EC00811=-138.9583,0.0000
EC00812=-136.5366,0.0000
EC00813=-135.0000,0.0000
EC00814=-133.4634,0.0000
EC00815=-131.0417,0.0000
EC00816=-127.9674,0.0000
EC00817=-127.2322,0.0000
EC00818=-127.3085,0.0000
EC00819=-127.4027,0.0000
EC00820=-127.4553,0.0000
EC00821=-127.3659,0.0000
EC00822=-125.6434,0.0000
EC00823=-122.6119,0.0000
EC00824=-118.7938,0.0000
EC00825=-114.6278,0.0000
EC00826=-110.3718,0.0000
EC00827=-106.2065,0.0000
EC00828=-102.3884,0.0000
EC00829=-99.3569,0.0000
EC00830=-97.6343,0.0000
EC00831=-97.5446,0.0000
EC00832=-97.5966,0.0000
EC00833=-97.6919,0.0000
EC00834=-97.7683,0.0000
EC00835=-97.0327,0.0000
EC00836=-93.9586,0.0000
EC00837=-91.5376,0.0000
EC00838=-90.0000,0.0000
EC00839=-88.4635,0.0000
EC00840=-86.0414,0.0000
EC00841=-82.9673,0.0000
EC00842=-82.2317,0.0000
EC00843=-82.3081,0.0000
EC00844=-82.4034,0.0000
EC00845=-82.4554,0.0000
EC00846=-82.3657,0.0000
EC00847=-80.6431,0.0000
EC00848=-77.6116,0.0000
EC00849=-73.7935,0.0000
EC00850=-69.6282,0.0000
EC00851=-65.3722,0.0000
EC00852=-61.2062,0.0000
EC00853=-57.3881,0.0000
EC00854=-54.3566,0.0000
EC00855=-52.6341,0.0000
EC00856=-52.5447,0.0000
EC00857=-52.5973,0.0000
EC00858=-52.6915,0.0000
EC00859=-52.7678,0.0000
EC00860=-52.0326,0.0000
EC00861=-48.9583,0.0000
EC00862=-46.5366,0.0000
EC00863=-45.0000,0.0000
EC00864=-43.4634,0.0000
EC00865=-41.0417,0.0000
EC00866=-37.9674,0.0000
EC00867=-37.2322,0.0000
EC00868=-37.3085,0.0000
EC00869=-37.4027,0.0000
EC00870=-37.4553,0.0000
EC00871=-37.3659,0.0000
EC00872=-35.6434,0.0000
EC00873=-32.6119,0.0000
EC00874=-28.7938,0.0000
EC00875=-24.6278,0.0000
EC00876=-20.3718,0.0000
EC00877=-16.2065,0.0000
EC00878=-12.3884,0.0000
EC00879=-9.3569,0.0000
EC00880=-7.6343,0.0000
EC00881=-7.5446,0.0000
EC00882=-7.5966,0.0000
EC00883=-7.6919,0.0000
EC00884=-7.7683,0.0000
EC00885=-7.0327,0.0000
EC00886=-3.9586,0.0000
EC00887=-1.5365,0.0000
EC00888=0.0000,0.0000
EC00889=0.0000,0.0000
EC00890=1.4747,0.0000
EC00891=3.8756,0.0000
EC00892=6.9699,0.0000
EC00893=7.6906,0.0000
EC00894=7.6170,0.0000
EC00895=7.5429,0.0000
EC00896=7.5106,0.0000
EC00897=7.6094,0.0000
EC00898=9.3401,0.0000
EC00899=35.6602,0.0000
EC00900=37.3910,0.0000
EC00901=37.4898,0.0000
EC00902=37.4572,0.0000
EC00903=37.3834,0.0000
EC00904=37.3085,0.0000
EC00905=38.0296,0.0000
EC00906=41.1238,0.0000
EC00907=43.5256,0.0000
EC00908=45.0000,0.0000
EC00909=46.4744,0.0000
EC00910=48.8762,0.0000
EC00911=51.9704,0.0000
EC00912=52.6915,0.0000
EC00913=52.6166,0.0000
EC00914=52.5428,0.0000
EC00915=52.5102,0.0000
EC00916=52.6090,0.0000
EC00917=54.3398,0.0000
EC00918=80.6599,0.0000
EC00919=82.3906,0.0000
EC00920=82.4894,0.0000
EC00921=82.4571,0.0000
EC00922=82.3830,0.0000
EC00923=82.3094,0.0000
EC00924=83.0301,0.0000
EC00925=86.1244,0.0000
EC00926=88.5253,0.0000
EC00927=90.0000,0.0000
EC00928=91.4736,0.0000
EC00929=93.8767,0.0000
EC00930=96.9699,0.0000
EC00931=97.6906,0.0000
EC00932=97.6170,0.0000
EC00933=97.5429,0.0000
EC00934=97.5106,0.0000
EC00935=97.6094,0.0000
EC00936=99.3401,0.0000
EC00937=125.6602,0.0000
EC00938=127.3910,0.0000
EC00939=127.4898,0.0000
EC00940=127.4572,0.0000
EC00941=127.3834,0.0000
EC00942=127.3085,0.0000
EC00943=128.0296,0.0000
EC00944=131.1238,0.0000
EC00945=133.5256,0.0000
EC00946=135.0000,0.0000
EC00947=136.4744,0.0000
EC00948=138.8762,0.0000
EC00949=141.9704,0.0000
EC00950=142.6915,0.0000
EC00951=142.6166,0.0000
EC00952=142.5428,0.0000
EC00953=142.5102,0.0000
EC00954=142.6090,0.0000
EC00955=144.3398,0.0000
EC00956=170.6599,0.0000
EC00957=172.3906,0.0000
EC00958=172.4894,0.0000
EC00959=172.4571,0.0000
EC00960=172.3830,0.0000
EC00961=172.3094,0.0000
EC00962=173.0301,0.0000
EC00963=176.1244,0.0000
EC00964=178.5253,0.0000
EC00965=180.0000,0.0000
EC00966=180.0000,0.0000
EC00967=-178.5264,0.0000
EC00968=-176.1233,0.0000
EC00969=-173.0301,0.0000
EC00970=-172.3094,0.0000
EC00971=-172.3830,0.0000
EC00972=-172.4571,0.0000
EC00973=-172.4894,0.0000
EC00974=-172.3906,0.0000
EC00975=-170.6599,0.0000
EC00976=-144.3398,0.0000
EC00977=-142.6090,0.0000
EC00978=-142.5102,0.0000
EC00979=-142.5428,0.0000
EC00980=-142.6166,0.0000
EC00981=-142.6915,0.0000
EC00982=-141.9704,0.0000
EC00983=-138.8762,0.0000
EC00984=-136.4744,0.0000
EC00985=-135.0000,0.0000
EC00986=-133.5256,0.0000
EC00987=-131.1238,0.0000
EC00988=-128.0296,0.0000
EC00989=-127.3085,0.0000
EC00990=-127.3834,0.0000
EC00991=-127.4572,0.0000
EC00992=-127.4898,0.0000
EC00993=-127.3910,0.0000
EC00994=-125.6602,0.0000
EC00995=-99.3401,0.0000
EC00996=-97.6094,0.0000
EC00997=-97.5106,0.0000
EC00998=-97.5429,0.0000
EC00999=-97.6170,0.0000
EC01000=-97.6906,0.0000
EC01001=-96.9699,0.0000
EC01002=-93.8756,0.0000
EC01003=-91.4747,0.0000
EC01004=-90.0000,0.0000
EC01005=-88.5264,0.0000
EC01006=-86.1233,0.0000
EC01007=-83.0301,0.0000
EC01008=-82.3094,0.0000
EC01009=-82.3830,0.0000
EC01010=-82.4571,0.0000
EC01011=-82.4894,0.0000
EC01012=-82.3906,0.0000
EC01013=-80.6599,0.0000
EC01014=-54.3398,0.0000
EC01015=-52.6090,0.0000
EC01016=-52.5102,0.0000
EC01017=-52.5428,0.0000
EC01018=-52.6166,0.0000
EC01019=-52.6915,0.0000
EC01020=-51.9704,0.0000
EC01021=-48.8762,0.0000
EC01022=-46.4744,0.0000
EC01023=-45.0000,0.0000
EC01024=-43.5256,0.0000
EC01025=-41.1238,0.0000
EC01026=-38.0296,0.0000
EC01027=-37.3085,0.0000
EC01028=-37.3834,0.0000
EC01029=-37.4572,0.0000
EC01030=-37.4898,0.0000
EC01031=-37.3910,0.0000
EC01032=-35.6602,0.0000
EC01033=-9.3401,0.0000
EC01034=-7.6094,0.0000
EC01035=-7.5106,0.0000
EC01036=-7.5429,0.0000
EC01037=-7.6170,0.0000
EC01038=-7.6906,0.0000
EC01039=-6.9699,0.0000
EC01040=-3.8767,0.0000
EC01041=-1.4736,0.0000
EC01042=0.0000,0.0000
EC01043=0.0000,0.0000
EC01044=1.4165,0.0000
EC01045=3.7994,0.0000
EC01046=6.9134,0.0000
EC01047=7.6249,0.0000
EC01048=7.5584,0.0000
EC01049=7.5104,0.0000
EC01050=37.4901,0.0000
EC01051=37.4412,0.0000
EC01052=37.3752,0.0000
EC01053=38.0867,0.0000
EC01054=41.2006,0.0000
EC01055=43.5844,0.0000
EC01056=45.0000,0.0000
EC01057=46.4156,0.0000
EC01058=48.8001,0.0000
EC01059=51.9133,0.0000
EC01060=52.6248,0.0000
EC01061=52.5588,0.0000
EC01062=52.5099,0.0000
EC01063=82.4896,0.0000
EC01064=82.4416,0.0000
EC01065=82.3751,0.0000
EC01066=83.0866,0.0000
EC01067=86.2006,0.0000
EC01068=88.5835,0.0000
EC01069=90.0000,0.0000
EC01070=91.4153,0.0000
EC01071=93.8005,0.0000
EC01072=96.9134,0.0000
EC01073=97.6249,0.0000
EC01074=97.5584,0.0000
EC01075=97.5104,0.0000
EC01076=127.4901,0.0000
EC01077=127.4412,0.0000
EC01078=127.3752,0.0000
EC01079=128.0867,0.0000
EC01080=131.2006,0.0000
EC01081=133.5844,0.0000
EC01082=135.0000,0.0000
EC01083=136.4156,0.0000
EC01084=138.8001,0.0000
EC01085=141.9133,0.0000
EC01086=142.6248,0.0000
EC01087=142.5588,0.0000
EC01088=142.5099,0.0000
EC01089=172.4896,0.0000
EC01090=172.4416,0.0000
EC01091=172.3751,0.0000
EC01092=173.0866,0.0000
EC01093=176.2006,0.0000
EC01094=178.5835,0.0000
EC01095=180.0000,0.0000
EC01096=180.0000,0.0000
EC01097=-178.5847,0.0000
EC01098=-176.1995,0.0000
EC01099=-173.0866,0.0000
EC01100=-172.3751,0.0000
EC01101=-172.4416,0.0000
EC01102=-172.4896,0.0000
EC01103=-142.5099,0.0000
EC01104=-142.5588,0.0000
EC01105=-142.6248,0.0000
EC01106=-141.9133,0.0000
EC01107=-138.7994,0.0000
EC01108=-136.4156,0.0000
EC01109=-135.0000,0.0000
EC01110=-133.5844,0.0000
EC01111=-131.1999,0.0000
EC01112=-128.0867,0.0000
EC01113=-127.3752,0.0000
EC01114=-127.4412,0.0000
EC01115=-127.4901,0.0000
EC01116=-97.5104,0.0000
EC01117=-97.5584,0.0000
EC01118=-97.6249,0.0000
EC01119=-96.9134,0.0000
EC01120=-93.7994,0.0000
EC01121=-91.4165,0.0000
EC01122=-90.0000,0.0000
EC01123=-88.5847,0.0000
EC01124=-86.1995,0.0000
EC01125=-83.0866,0.0000
EC01126=-82.3751,0.0000
EC01127=-82.4416,0.0000
EC01128=-82.4896,0.0000
EC01129=-52.5099,0.0000
EC01130=-52.5588,0.0000
EC01131=-52.6248,0.0000
EC01132=-51.9133,0.0000
EC01133=-48.7994,0.0000
EC01134=-46.4156,0.0000
EC01135=-45.0000,0.0000
EC01136=-43.5844,0.0000
EC01137=-41.1999,0.0000
EC01138=-38.0867,0.0000
EC01139=-37.3752,0.0000
EC01140=-37.4412,0.0000
EC01141=-37.4901,0.0000
EC01142=-7.5104,0.0000
EC01143=-7.5584,0.0000
EC01144=-7.6249,0.0000
EC01145=-6.9134,0.0000
EC01146=-3.8005,0.0000
EC01147=-1.4153,0.0000
EC01148=0.0000,0.0000
EC01149=0.0000,0.0000
EC01150=1.3641,0.0000
EC01151=3.7307,0.0000
EC01152=6.8641,0.0000
EC01153=7.5707,0.0000
EC01154=7.5193,0.0000
EC01155=37.4799,0.0000
EC01156=37.4296,0.0000
EC01157=38.1360,0.0000
EC01158=41.2692,0.0000
EC01159=43.6362,0.0000
EC01160=45.0000,0.0000
EC01161=46.3630,0.0000
EC01162=48.7308,0.0000
EC01163=51.8640,0.0000
EC01164=52.5704,0.0000
EC01165=52.5201,0.0000
EC01166=82.4807,0.0000
EC01167=82.4293,0.0000
EC01168=83.1359,0.0000
EC01169=86.2693,0.0000
EC01170=88.6359,0.0000
EC01171=90.0000,0.0000
EC01172=91.3630,0.0000
EC01173=93.7318,0.0000
EC01174=96.8641,0.0000
EC01175=97.5707,0.0000
EC01176=97.5193,0.0000
EC01177=127.4799,0.0000
EC01178=127.4296,0.0000
EC01179=128.1360,0.0000
EC01180=131.2692,0.0000
EC01181=133.6362,0.0000
EC01182=135.0000,0.0000
EC01183=136.3630,0.0000
EC01184=138.7308,0.0000
EC01185=141.8640,0.0000
EC01186=142.5704,0.0000
EC01187=142.5201,0.0000
EC01188=172.4807,0.0000
EC01189=172.4293,0.0000
EC01190=173.1359,0.0000
EC01191=176.2693,0.0000
EC01192=178.6359,0.0000
EC01193=180.0000,0.0000
EC01194=180.0000,0.0000
EC01195=-178.6370,0.0000
EC01196=-176.2682,0.0000
EC01197=-173.1359,0.0000
EC01198=-172.4293,0.0000
EC01199=-172.4807,0.0000
EC01200=-142.5201,0.0000
EC01201=-142.5704,0.0000
EC01202=-141.8640,0.0000
EC01203=-138.7308,0.0000
EC01204=-136.3638,0.0000
EC01205=-135.0000,0.0000
EC01206=-133.6370,0.0000
EC01207=-131.2692,0.0000
EC01208=-128.1360,0.0000
EC01209=-127.4296,0.0000
EC01210=-127.4799,0.0000
EC01211=-97.5193,0.0000
EC01212=-97.5707,0.0000
EC01213=-96.8641,0.0000
EC01214=-93.7307,0.0000
EC01215=-91.3641,0.0000
EC01216=-90.0000,0.0000
EC01217=-88.6370,0.0000
EC01218=-86.2682,0.0000
EC01219=-83.1359,0.0000
EC01220=-82.4293,0.0000
EC01221=-82.4807,0.0000
EC01222=-52.5201,0.0000
EC01223=-52.5704,0.0000
EC01224=-51.8640,0.0000
EC01225=-48.7308,0.0000
EC01226=-46.3638,0.0000
EC01227=-45.0000,0.0000
EC01228=-43.6370,0.0000
EC01229=-41.2692,0.0000
EC01230=-38.1360,0.0000
EC01231=-37.4296,0.0000
EC01232=-37.4799,0.0000
EC01233=-7.5193,0.0000
EC01234=-7.5707,0.0000
EC01235=-6.8641,0.0000
EC01236=-3.7318,0.0000
EC01237=-1.3630,0.0000
EC01238=0.0000,0.0000
EC01239=0.0000,0.0000
EC01240=1.3191,0.0000
EC01241=3.6720,0.0000
EC01242=6.8225,0.0000
EC01243=7.5303,0.0000
EC01244=7.5014,0.0000
EC01245=37.4983,0.0000
EC01246=37.4688,0.0000
EC01247=38.1772,0.0000
EC01248=41.3279,0.0000
EC01249=43.6816,0.0000
EC01250=45.0000,0.0000
EC01251=46.3184,0.0000
EC01252=48.6728,0.0000
EC01253=51.8228,0.0000
EC01254=52.5312,0.0000
EC01255=52.5017,0.0000
EC01256=82.4986,0.0000
EC01257=82.4697,0.0000
EC01258=83.1775,0.0000
EC01259=86.3280,0.0000
EC01260=88.6809,0.0000
EC01261=90.0000,0.0000
EC01262=91.3180,0.0000
EC01263=93.6719,0.0000
EC01264=96.8225,0.0000
EC01265=97.5303,0.0000
EC01266=97.5014,0.0000
EC01267=127.4983,0.0000
EC01268=127.4688,0.0000
EC01269=128.1772,0.0000
EC01270=131.3279,0.0000
EC01271=133.6816,0.0000
EC01272=135.0000,0.0000
EC01273=136.3184,0.0000
EC01274=138.6728,0.0000
EC01275=141.8228,0.0000
EC01276=142.5312,0.0000
EC01277=142.5017,0.0000
EC01278=172.4986,0.0000
EC01279=172.4697,0.0000
EC01280=173.1775,0.0000
EC01281=176.3280,0.0000
EC01282=178.6809,0.0000
EC01283=180.0000,0.0000
EC01284=180.0000,0.0000
EC01285=-178.6820,0.0000
EC01286=-176.3281,0.0000
EC01287=-173.1775,0.0000
EC01288=-172.4697,0.0000
EC01289=-172.4986,0.0000
EC01290=-142.5017,0.0000
EC01291=-142.5312,0.0000
EC01292=-141.8228,0.0000
EC01293=-138.6721,0.0000
EC01294=-136.3184,0.0000
EC01295=-135.0000,0.0000
EC01296=-133.6816,0.0000
EC01297=-131.3272,0.0000
EC01298=-128.1772,0.0000
EC01299=-127.4688,0.0000
EC01300=-127.4983,0.0000
EC01301=-97.5014,0.0000
EC01302=-97.5303,0.0000
EC01303=-96.8225,0.0000
EC01304=-93.6720,0.0000
EC01305=-91.3191,0.0000
EC01306=-90.0000,0.0000
EC01307=-88.6820,0.0000
EC01308=-86.3281,0.0000
EC01309=-83.1775,0.0000
EC01310=-82.4697,0.0000
EC01311=-82.4986,0.0000
EC01312=-52.5017,0.0000
EC01313=-52.5312,0.0000
EC01314=-51.8228,0.0000
EC01315=-48.6721,0.0000
EC01316=-46.3184,0.0000
EC01317=-45.0000,0.0000
EC01318=-43.6816,0.0000
EC01319=-41.3272,0.0000
EC01320=-38.1772,0.0000
EC01321=-37.4688,0.0000
EC01322=-37.4983,0.0000
EC01323=-7.5014,0.0000
EC01324=-7.5303,0.0000
EC01325=-6.8225,0.0000
EC01326=-3.6719,0.0000
EC01327=-1.3180,0.0000
EC01328=0.0000,0.0000
EC01329=0.0000,0.0000
EC01330=1.2828,0.0000
EC01331=3.6251,0.0000
EC01332=6.7919,0.0000
EC01333=7.5071,0.0000
EC01334=37.4934,0.0000
EC01335=38.2087,0.0000
EC01336=41.3754,0.0000
EC01337=43.7178,0.0000
EC01338=45.0000,0.0000
EC01339=46.2813,0.0000
EC01340=48.6253,0.0000
EC01341=51.7913,0.0000
EC01342=52.5066,0.0000
EC01343=82.4929,0.0000
EC01344=83.2081,0.0000
EC01345=86.3749,0.0000
EC01346=88.7172,0.0000
EC01347=90.0000,0.0000
EC01348=91.2817,0.0000
EC01349=93.6251,0.0000
EC01350=96.7919,0.0000
EC01351=97.5071,0.0000
EC01352=127.4934,0.0000
EC01353=128.2087,0.0000
EC01354=131.3754,0.0000
EC01355=133.7178,0.0000
EC01356=135.0000,0.0000
EC01357=136.2813,0.0000
EC01358=138.6253,0.0000
EC01359=141.7913,0.0000
EC01360=142.5066,0.0000
EC01361=172.4929,0.0000
EC01362=173.2081,0.0000
EC01363=176.3749,0.0000
EC01364=178.7172,0.0000
EC01365=180.0000,0.0000
EC01366=180.0000,0.0000
EC01367=-178.7183,0.0000
EC01368=-176.3749,0.0000
EC01369=-173.2081,0.0000
EC01370=-172.4929,0.0000
EC01371=-142.5066,0.0000
EC01372=-141.7913,0.0000
EC01373=-138.6246,0.0000
EC01374=-136.2822,0.0000
EC01375=-135.0000,0.0000
EC01376=-133.7187,0.0000
EC01377=-131.3747,0.0000
EC01378=-128.2087,0.0000
EC01379=-127.4934,0.0000
EC01380=-97.5071,0.0000
EC01381=-96.7919,0.0000
EC01382=-93.6251,0.0000
EC01383=-91.2828,0.0000
EC01384=-90.0000,0.0000
EC01385=-88.7183,0.0000
EC01386=-86.3749,0.0000
EC01387=-83.2081,0.0000
EC01388=-82.4929,0.0000
EC01389=-52.5066,0.0000
EC01390=-51.7913,0.0000
EC01391=-48.6246,0.0000
EC01392=-46.2822,0.0000
EC01393=-45.0000,0.0000
EC01394=-43.7187,0.0000
EC01395=-41.3747,0.0000
EC01396=-38.2087,0.0000
EC01397=-37.4934,0.0000
EC01398=-7.5071,0.0000
EC01399=-6.7919,0.0000
EC01400=-3.6251,0.0000
EC01401=-1.2817,0.0000
EC01402=0.0000,0.0000
EC01403=0.0000,0.0000
EC01404=1.2567,0.0000
EC01405=3.5913,0.0000
EC01406=6.7714,0.0000
EC01407=38.2287,0.0000
EC01408=41.4086,0.0000
EC01409=43.7431,0.0000
EC01410=45.0000,0.0000
EC01411=46.2560,0.0000
EC01412=48.5914,0.0000
EC01413=51.7713,0.0000
EC01414=83.2286,0.0000
EC01415=86.4087,0.0000
EC01416=88.7433,0.0000
EC01417=90.0000,0.0000
EC01418=91.2567,0.0000
EC01419=93.5913,0.0000
EC01420=96.7713,0.0000
EC01421=128.2287,0.0000
EC01422=131.4086,0.0000
EC01423=133.7431,0.0000
EC01424=135.0000,0.0000
EC01425=136.2560,0.0000
EC01426=138.5914,0.0000
EC01427=141.7713,0.0000
EC01428=173.2286,0.0000
EC01429=176.4087,0.0000
EC01430=178.7433,0.0000
EC01431=180.0000,0.0000
EC01432=180.0000,0.0000
EC01433=-178.7433,0.0000
EC01434=-176.4087,0.0000
EC01435=-173.2287,0.0000
EC01436=-141.7713,0.0000
EC01437=-138.5914,0.0000
EC01438=-136.2569,0.0000
EC01439=-135.0000,0.0000
EC01440=-133.7440,0.0000
EC01441=-131.4086,0.0000
EC01442=-128.2287,0.0000
EC01443=-96.7714,0.0000
EC01444=-93.5913,0.0000
EC01445=-91.2567,0.0000
EC01446=-90.0000,0.0000
EC01447=-88.7433,0.0000
EC01448=-86.4087,0.0000
EC01449=-83.2287,0.0000
EC01450=-51.7713,0.0000
EC01451=-48.5914,0.0000
EC01452=-46.2569,0.0000
EC01453=-45.0000,0.0000
EC01454=-43.7440,0.0000
EC01455=-41.4086,0.0000
EC01456=-38.2287,0.0000
EC01457=-6.7713,0.0000
EC01458=-3.5913,0.0000
EC01459=-1.2567,0.0000
EC01460=0.0000,0.0000
EC01461=0.0000,0.0000
EC01462=1.2432,0.0000
EC01463=3.5737,0.0000
EC01464=6.7645,0.0000
EC01465=38.2351,0.0000
EC01466=41.4267,0.0000
EC01467=43.7573,0.0000
EC01468=45.0000,0.0000
EC01469=46.2427,0.0000
EC01470=48.5742,0.0000
EC01471=51.7649,0.0000
EC01472=83.2355,0.0000
EC01473=86.4263,0.0000
EC01474=88.7568,0.0000
EC01475=90.0000,0.0000
EC01476=91.2420,0.0000
EC01477=93.5737,0.0000
EC01478=96.7645,0.0000
EC01479=128.2351,0.0000
EC01480=131.4267,0.0000
EC01481=133.7573,0.0000
EC01482=135.0000,0.0000
EC01483=136.2427,0.0000
EC01484=138.5742,0.0000
EC01485=141.7649,0.0000
EC01486=173.2355,0.0000
EC01487=176.4263,0.0000
EC01488=178.7568,0.0000
EC01489=180.0000,0.0000
EC01490=180.0000,0.0000
EC01491=-178.7580,0.0000
EC01492=-176.4263,0.0000
EC01493=-173.2355,0.0000
EC01494=-141.7649,0.0000
EC01495=-138.5733,0.0000
EC01496=-136.2427,0.0000
EC01497=-135.0000,0.0000
EC01498=-133.7573,0.0000
EC01499=-131.4258,0.0000
EC01500=-128.2351,0.0000
EC01501=-96.7645,0.0000
EC01502=-93.5737,0.0000
EC01503=-91.2432,0.0000
EC01504=-90.0000,0.0000
EC01505=-88.7580,0.0000
EC01506=-86.4263,0.0000
EC01507=-83.2355,0.0000
EC01508=-51.7649,0.0000
EC01509=-48.5733,0.0000
EC01510=-46.2427,0.0000
EC01511=-45.0000,0.0000
EC01512=-43.7573,0.0000
EC01513=-41.4258,0.0000
EC01514=-38.2351,0.0000
EC01515=-6.7645,0.0000
EC01516=-3.5737,0.0000
EC01517=-1.2420,0.0000
EC01518=0.0000,0.0000
//INST
///DATE 2021/02/10 13:51
///COMM
///ATTR SC,RW,RJ
////FRAME USER 2
///GROUP1 RB1
///GROUP2 ST1
NOP
SMOVL C00000 +MOVJ EC00000
SMOVL C00001 +MOVJ EC00001
SMOVL C00002 +MOVJ EC00002
SMOVL C00003 +MOVJ EC00003
SMOVL C00004 +MOVJ EC00004
SMOVL C00005 +MOVJ EC00005
SMOVL C00006 +MOVJ EC00006
SMOVL C00007 +MOVJ EC00007
SMOVL C00008 +MOVJ EC00008
SMOVL C00009 +MOVJ EC00009
SMOVL C00010 +MOVJ EC00010
SMOVL C00011 +MOVJ EC00011
SMOVL C00012 +MOVJ EC00012
SMOVL C00013 +MOVJ EC00013
SMOVL C00014 +MOVJ EC00014
SMOVL C00015 +MOVJ EC00015
SMOVL C00016 +MOVJ EC00016
SMOVL C00017 +MOVJ EC00017
SMOVL C00018 +MOVJ EC00018
SMOVL C00019 +MOVJ EC00019
SMOVL C00020 +MOVJ EC00020
SMOVL C00021 +MOVJ EC00021
SMOVL C00022 +MOVJ EC00022
SMOVL C00023 +MOVJ EC00023
SMOVL C00024 +MOVJ EC00024
SMOVL C00025 +MOVJ EC00025
SMOVL C00026 +MOVJ EC00026
SMOVL C00027 +MOVJ EC00027
SMOVL C00028 +MOVJ EC00028
SMOVL C00029 +MOVJ EC00029
SMOVL C00030 +MOVJ EC00030
SMOVL C00031 +MOVJ EC00031
SMOVL C00032 +MOVJ EC00032
SMOVL C00033 +MOVJ EC00033
SMOVL C00034 +MOVJ EC00034
SMOVL C00035 +MOVJ EC00035
SMOVL C00036 +MOVJ EC00036
SMOVL C00037 +MOVJ EC00037
SMOVL C00038 +MOVJ EC00038
SMOVL C00039 +MOVJ EC00039
SMOVL C00040 +MOVJ EC00040
SMOVL C00041 +MOVJ EC00041
SMOVL C00042 +MOVJ EC00042
SMOVL C00043 +MOVJ EC00043
SMOVL C00044 +MOVJ EC00044
SMOVL C00045 +MOVJ EC00045
SMOVL C00046 +MOVJ EC00046
SMOVL C00047 +MOVJ EC00047
SMOVL C00048 +MOVJ EC00048
SMOVL C00049 +MOVJ EC00049
SMOVL C00050 +MOVJ EC00050
SMOVL C00051 +MOVJ EC00051
SMOVL C00052 +MOVJ EC00052
SMOVL C00053 +MOVJ EC00053
SMOVL C00054 +MOVJ EC00054
SMOVL C00055 +MOVJ EC00055
SMOVL C00056 +MOVJ EC00056
SMOVL C00057 +MOVJ EC00057
SMOVL C00058 +MOVJ EC00058
SMOVL C00059 +MOVJ EC00059
SMOVL C00060 +MOVJ EC00060
SMOVL C00061 +MOVJ EC00061
SMOVL C00062 +MOVJ EC00062
SMOVL C00063 +MOVJ EC00063
SMOVL C00064 +MOVJ EC00064
SMOVL C00065 +MOVJ EC00065
SMOVL C00066 +MOVJ EC00066
SMOVL C00067 +MOVJ EC00067
SMOVL C00068 +MOVJ EC00068
SMOVL C00069 +MOVJ EC00069
SMOVL C00070 +MOVJ EC00070
SMOVL C00071 +MOVJ EC00071
SMOVL C00072 +MOVJ EC00072
SMOVL C00073 +MOVJ EC00073
SMOVL C00074 +MOVJ EC00074
SMOVL C00075 +MOVJ EC00075
SMOVL C00076 +MOVJ EC00076
SMOVL C00077 +MOVJ EC00077
SMOVL C00078 +MOVJ EC00078
SMOVL C00079 +MOVJ EC00079
SMOVL C00080 +MOVJ EC00080
SMOVL C00081 +MOVJ EC00081
SMOVL C00082 +MOVJ EC00082
SMOVL C00083 +MOVJ EC00083
SMOVL C00084 +MOVJ EC00084
SMOVL C00085 +MOVJ EC00085
SMOVL C00086 +MOVJ EC00086
SMOVL C00087 +MOVJ EC00087
SMOVL C00088 +MOVJ EC00088
SMOVL C00089 +MOVJ EC00089
SMOVL C00090 +MOVJ EC00090
SMOVL C00091 +MOVJ EC00091
SMOVL C00092 +MOVJ EC00092
SMOVL C00093 +MOVJ EC00093
SMOVL C00094 +MOVJ EC00094
SMOVL C00095 +MOVJ EC00095
SMOVL C00096 +MOVJ EC00096
SMOVL C00097 +MOVJ EC00097
SMOVL C00098 +MOVJ EC00098
SMOVL C00099 +MOVJ EC00099
SMOVL C00100 +MOVJ EC00100
SMOVL C00101 +MOVJ EC00101
SMOVL C00102 +MOVJ EC00102
SMOVL C00103 +MOVJ EC00103
SMOVL C00104 +MOVJ EC00104
SMOVL C00105 +MOVJ EC00105
SMOVL C00106 +MOVJ EC00106
SMOVL C00107 +MOVJ EC00107
SMOVL C00108 +MOVJ EC00108
SMOVL C00109 +MOVJ EC00109
SMOVL C00110 +MOVJ EC00110
SMOVL C00111 +MOVJ EC00111
SMOVL C00112 +MOVJ EC00112
SMOVL C00113 +MOVJ EC00113
SMOVL C00114 +MOVJ EC00114
SMOVL C00115 +MOVJ EC00115
SMOVL C00116 +MOVJ EC00116
SMOVL C00117 +MOVJ EC00117
SMOVL C00118 +MOVJ EC00118
SMOVL C00119 +MOVJ EC00119
SMOVL C00120 +MOVJ EC00120
SMOVL C00121 +MOVJ EC00121
SMOVL C00122 +MOVJ EC00122
SMOVL C00123 +MOVJ EC00123
SMOVL C00124 +MOVJ EC00124
SMOVL C00125 +MOVJ EC00125
SMOVL C00126 +MOVJ EC00126
SMOVL C00127 +MOVJ EC00127
SMOVL C00128 +MOVJ EC00128
SMOVL C00129 +MOVJ EC00129
SMOVL C00130 +MOVJ EC00130
SMOVL C00131 +MOVJ EC00131
SMOVL C00132 +MOVJ EC00132
SMOVL C00133 +MOVJ EC00133
SMOVL C00134 +MOVJ EC00134
SMOVL C00135 +MOVJ EC00135
SMOVL C00136 +MOVJ EC00136
SMOVL C00137 +MOVJ EC00137
SMOVL C00138 +MOVJ EC00138
SMOVL C00139 +MOVJ EC00139
SMOVL C00140 +MOVJ EC00140
SMOVL C00141 +MOVJ EC00141
SMOVL C00142 +MOVJ EC00142
SMOVL C00143 +MOVJ EC00143
SMOVL C00144 +MOVJ EC00144
SMOVL C00145 +MOVJ EC00145
SMOVL C00146 +MOVJ EC00146
SMOVL C00147 +MOVJ EC00147
SMOVL C00148 +MOVJ EC00148
SMOVL C00149 +MOVJ EC00149
SMOVL C00150 +MOVJ EC00150
SMOVL C00151 +MOVJ EC00151
SMOVL C00152 +MOVJ EC00152
SMOVL C00153 +MOVJ EC00153
SMOVL C00154 +MOVJ EC00154
SMOVL C00155 +MOVJ EC00155
SMOVL C00156 +MOVJ EC00156
SMOVL C00157 +MOVJ EC00157
SMOVL C00158 +MOVJ EC00158
SMOVL C00159 +MOVJ EC00159
SMOVL C00160 +MOVJ EC00160
SMOVL C00161 +MOVJ EC00161
SMOVL C00162 +MOVJ EC00162
SMOVL C00163 +MOVJ EC00163
SMOVL C00164 +MOVJ EC00164
SMOVL C00165 +MOVJ EC00165
SMOVL C00166 +MOVJ EC00166
SMOVL C00167 +MOVJ EC00167
SMOVL C00168 +MOVJ EC00168
SMOVL C00169 +MOVJ EC00169
SMOVL C00170 +MOVJ EC00170
SMOVL C00171 +MOVJ EC00171
SMOVL C00172 +MOVJ EC00172
SMOVL C00173 +MOVJ EC00173
SMOVL C00174 +MOVJ EC00174
SMOVL C00175 +MOVJ EC00175
SMOVL C00176 +MOVJ EC00176
SMOVL C00177 +MOVJ EC00177
SMOVL C00178 +MOVJ EC00178
SMOVL C00179 +MOVJ EC00179
SMOVL C00180 +MOVJ EC00180
SMOVL C00181 +MOVJ EC00181
SMOVL C00182 +MOVJ EC00182
SMOVL C00183 +MOVJ EC00183
SMOVL C00184 +MOVJ EC00184
SMOVL C00185 +MOVJ EC00185
SMOVL C00186 +MOVJ EC00186
SMOVL C00187 +MOVJ EC00187
SMOVL C00188 +MOVJ EC00188
SMOVL C00189 +MOVJ EC00189
SMOVL C00190 +MOVJ EC00190
SMOVL C00191 +MOVJ EC00191
SMOVL C00192 +MOVJ EC00192
SMOVL C00193 +MOVJ EC00193
SMOVL C00194 +MOVJ EC00194
SMOVL C00195 +MOVJ EC00195
SMOVL C00196 +MOVJ EC00196
SMOVL C00197 +MOVJ EC00197
SMOVL C00198 +MOVJ EC00198
SMOVL C00199 +MOVJ EC00199
SMOVL C00200 +MOVJ EC00200
SMOVL C00201 +MOVJ EC00201
SMOVL C00202 +MOVJ EC00202
SMOVL C00203 +MOVJ EC00203
SMOVL C00204 +MOVJ EC00204
SMOVL C00205 +MOVJ EC00205
SMOVL C00206 +MOVJ EC00206
SMOVL C00207 +MOVJ EC00207
SMOVL C00208 +MOVJ EC00208
SMOVL C00209 +MOVJ EC00209
SMOVL C00210 +MOVJ EC00210
SMOVL C00211 +MOVJ EC00211
SMOVL C00212 +MOVJ EC00212
SMOVL C00213 +MOVJ EC00213
SMOVL C00214 +MOVJ EC00214
SMOVL C00215 +MOVJ EC00215
SMOVL C00216 +MOVJ EC00216
SMOVL C00217 +MOVJ EC00217
SMOVL C00218 +MOVJ EC00218
SMOVL C00219 +MOVJ EC00219
SMOVL C00220 +MOVJ EC00220
SMOVL C00221 +MOVJ EC00221
SMOVL C00222 +MOVJ EC00222
SMOVL C00223 +MOVJ EC00223
SMOVL C00224 +MOVJ EC00224
SMOVL C00225 +MOVJ EC00225
SMOVL C00226 +MOVJ EC00226
SMOVL C00227 +MOVJ EC00227
SMOVL C00228 +MOVJ EC00228
SMOVL C00229 +MOVJ EC00229
SMOVL C00230 +MOVJ EC00230
SMOVL C00231 +MOVJ EC00231
SMOVL C00232 +MOVJ EC00232
SMOVL C00233 +MOVJ EC00233
SMOVL C00234 +MOVJ EC00234
SMOVL C00235 +MOVJ EC00235
SMOVL C00236 +MOVJ EC00236
SMOVL C00237 +MOVJ EC00237
SMOVL C00238 +MOVJ EC00238
SMOVL C00239 +MOVJ EC00239
SMOVL C00240 +MOVJ EC00240
SMOVL C00241 +MOVJ EC00241
SMOVL C00242 +MOVJ EC00242
SMOVL C00243 +MOVJ EC00243
SMOVL C00244 +MOVJ EC00244
SMOVL C00245 +MOVJ EC00245
SMOVL C00246 +MOVJ EC00246
SMOVL C00247 +MOVJ EC00247
SMOVL C00248 +MOVJ EC00248
SMOVL C00249 +MOVJ EC00249
SMOVL C00250 +MOVJ EC00250
SMOVL C00251 +MOVJ EC00251
SMOVL C00252 +MOVJ EC00252
SMOVL C00253 +MOVJ EC00253
SMOVL C00254 +MOVJ EC00254
SMOVL C00255 +MOVJ EC00255
SMOVL C00256 +MOVJ EC00256
SMOVL C00257 +MOVJ EC00257
SMOVL C00258 +MOVJ EC00258
SMOVL C00259 +MOVJ EC00259
SMOVL C00260 +MOVJ EC00260
SMOVL C00261 +MOVJ EC00261
SMOVL C00262 +MOVJ EC00262
SMOVL C00263 +MOVJ EC00263
SMOVL C00264 +MOVJ EC00264
SMOVL C00265 +MOVJ EC00265
SMOVL C00266 +MOVJ EC00266
SMOVL C00267 +MOVJ EC00267
SMOVL C00268 +MOVJ EC00268
SMOVL C00269 +MOVJ EC00269
SMOVL C00270 +MOVJ EC00270
SMOVL C00271 +MOVJ EC00271
SMOVL C00272 +MOVJ EC00272
SMOVL C00273 +MOVJ EC00273
SMOVL C00274 +MOVJ EC00274
SMOVL C00275 +MOVJ EC00275
SMOVL C00276 +MOVJ EC00276
SMOVL C00277 +MOVJ EC00277
SMOVL C00278 +MOVJ EC00278
SMOVL C00279 +MOVJ EC00279
SMOVL C00280 +MOVJ EC00280
SMOVL C00281 +MOVJ EC00281
SMOVL C00282 +MOVJ EC00282
SMOVL C00283 +MOVJ EC00283
SMOVL C00284 +MOVJ EC00284
SMOVL C00285 +MOVJ EC00285
SMOVL C00286 +MOVJ EC00286
SMOVL C00287 +MOVJ EC00287
SMOVL C00288 +MOVJ EC00288
SMOVL C00289 +MOVJ EC00289
SMOVL C00290 +MOVJ EC00290
SMOVL C00291 +MOVJ EC00291
SMOVL C00292 +MOVJ EC00292
SMOVL C00293 +MOVJ EC00293
SMOVL C00294 +MOVJ EC00294
SMOVL C00295 +MOVJ EC00295
SMOVL C00296 +MOVJ EC00296
SMOVL C00297 +MOVJ EC00297
SMOVL C00298 +MOVJ EC00298
SMOVL C00299 +MOVJ EC00299
SMOVL C00300 +MOVJ EC00300
SMOVL C00301 +MOVJ EC00301
SMOVL C00302 +MOVJ EC00302
SMOVL C00303 +MOVJ EC00303
SMOVL C00304 +MOVJ EC00304
SMOVL C00305 +MOVJ EC00305
SMOVL C00306 +MOVJ EC00306
SMOVL C00307 +MOVJ EC00307
SMOVL C00308 +MOVJ EC00308
SMOVL C00309 +MOVJ EC00309
SMOVL C00310 +MOVJ EC00310
SMOVL C00311 +MOVJ EC00311
SMOVL C00312 +MOVJ EC00312
SMOVL C00313 +MOVJ EC00313
SMOVL C00314 +MOVJ EC00314
SMOVL C00315 +MOVJ EC00315
SMOVL C00316 +MOVJ EC00316
SMOVL C00317 +MOVJ EC00317
SMOVL C00318 +MOVJ EC00318
SMOVL C00319 +MOVJ EC00319
SMOVL C00320 +MOVJ EC00320
SMOVL C00321 +MOVJ EC00321
SMOVL C00322 +MOVJ EC00322
SMOVL C00323 +MOVJ EC00323
SMOVL C00324 +MOVJ EC00324
SMOVL C00325 +MOVJ EC00325
SMOVL C00326 +MOVJ EC00326
SMOVL C00327 +MOVJ EC00327
SMOVL C00328 +MOVJ EC00328
SMOVL C00329 +MOVJ EC00329
SMOVL C00330 +MOVJ EC00330
SMOVL C00331 +MOVJ EC00331
SMOVL C00332 +MOVJ EC00332
SMOVL C00333 +MOVJ EC00333
SMOVL C00334 +MOVJ EC00334
SMOVL C00335 +MOVJ EC00335
SMOVL C00336 +MOVJ EC00336
SMOVL C00337 +MOVJ EC00337
SMOVL C00338 +MOVJ EC00338
SMOVL C00339 +MOVJ EC00339
SMOVL C00340 +MOVJ EC00340
SMOVL C00341 +MOVJ EC00341
SMOVL C00342 +MOVJ EC00342
SMOVL C00343 +MOVJ EC00343
SMOVL C00344 +MOVJ EC00344
SMOVL C00345 +MOVJ EC00345
SMOVL C00346 +MOVJ EC00346
SMOVL C00347 +MOVJ EC00347
SMOVL C00348 +MOVJ EC00348
SMOVL C00349 +MOVJ EC00349
SMOVL C00350 +MOVJ EC00350
SMOVL C00351 +MOVJ EC00351
SMOVL C00352 +MOVJ EC00352
SMOVL C00353 +MOVJ EC00353
SMOVL C00354 +MOVJ EC00354
SMOVL C00355 +MOVJ EC00355
SMOVL C00356 +MOVJ EC00356
SMOVL C00357 +MOVJ EC00357
SMOVL C00358 +MOVJ EC00358
SMOVL C00359 +MOVJ EC00359
SMOVL C00360 +MOVJ EC00360
SMOVL C00361 +MOVJ EC00361
SMOVL C00362 +MOVJ EC00362
SMOVL C00363 +MOVJ EC00363
SMOVL C00364 +MOVJ EC00364
SMOVL C00365 +MOVJ EC00365
SMOVL C00366 +MOVJ EC00366
SMOVL C00367 +MOVJ EC00367
SMOVL C00368 +MOVJ EC00368
SMOVL C00369 +MOVJ EC00369
SMOVL C00370 +MOVJ EC00370
SMOVL C00371 +MOVJ EC00371
SMOVL C00372 +MOVJ EC00372
SMOVL C00373 +MOVJ EC00373
SMOVL C00374 +MOVJ EC00374
SMOVL C00375 +MOVJ EC00375
SMOVL C00376 +MOVJ EC00376
SMOVL C00377 +MOVJ EC00377
SMOVL C00378 +MOVJ EC00378
SMOVL C00379 +MOVJ EC00379
SMOVL C00380 +MOVJ EC00380
SMOVL C00381 +MOVJ EC00381
SMOVL C00382 +MOVJ EC00382
SMOVL C00383 +MOVJ EC00383
SMOVL C00384 +MOVJ EC00384
SMOVL C00385 +MOVJ EC00385
SMOVL C00386 +MOVJ EC00386
SMOVL C00387 +MOVJ EC00387
SMOVL C00388 +MOVJ EC00388
SMOVL C00389 +MOVJ EC00389
SMOVL C00390 +MOVJ EC00390
SMOVL C00391 +MOVJ EC00391
SMOVL C00392 +MOVJ EC00392
SMOVL C00393 +MOVJ EC00393
SMOVL C00394 +MOVJ EC00394
SMOVL C00395 +MOVJ EC00395
SMOVL C00396 +MOVJ EC00396
SMOVL C00397 +MOVJ EC00397
SMOVL C00398 +MOVJ EC00398
SMOVL C00399 +MOVJ EC00399
SMOVL C00400 +MOVJ EC00400
SMOVL C00401 +MOVJ EC00401
SMOVL C00402 +MOVJ EC00402
SMOVL C00403 +MOVJ EC00403
SMOVL C00404 +MOVJ EC00404
SMOVL C00405 +MOVJ EC00405
SMOVL C00406 +MOVJ EC00406
SMOVL C00407 +MOVJ EC00407
SMOVL C00408 +MOVJ EC00408
SMOVL C00409 +MOVJ EC00409
SMOVL C00410 +MOVJ EC00410
SMOVL C00411 +MOVJ EC00411
SMOVL C00412 +MOVJ EC00412
SMOVL C00413 +MOVJ EC00413
SMOVL C00414 +MOVJ EC00414
SMOVL C00415 +MOVJ EC00415
SMOVL C00416 +MOVJ EC00416
SMOVL C00417 +MOVJ EC00417
SMOVL C00418 +MOVJ EC00418
SMOVL C00419 +MOVJ EC00419
SMOVL C00420 +MOVJ EC00420
SMOVL C00421 +MOVJ EC00421
SMOVL C00422 +MOVJ EC00422
SMOVL C00423 +MOVJ EC00423
SMOVL C00424 +MOVJ EC00424
SMOVL C00425 +MOVJ EC00425
SMOVL C00426 +MOVJ EC00426
SMOVL C00427 +MOVJ EC00427
SMOVL C00428 +MOVJ EC00428
SMOVL C00429 +MOVJ EC00429
SMOVL C00430 +MOVJ EC00430
SMOVL C00431 +MOVJ EC00431
SMOVL C00432 +MOVJ EC00432
SMOVL C00433 +MOVJ EC00433
SMOVL C00434 +MOVJ EC00434
SMOVL C00435 +MOVJ EC00435
SMOVL C00436 +MOVJ EC00436
SMOVL C00437 +MOVJ EC00437
SMOVL C00438 +MOVJ EC00438
SMOVL C00439 +MOVJ EC00439
SMOVL C00440 +MOVJ EC00440
SMOVL C00441 +MOVJ EC00441
SMOVL C00442 +MOVJ EC00442
SMOVL C00443 +MOVJ EC00443
SMOVL C00444 +MOVJ EC00444
SMOVL C00445 +MOVJ EC00445
SMOVL C00446 +MOVJ EC00446
SMOVL C00447 +MOVJ EC00447
SMOVL C00448 +MOVJ EC00448
SMOVL C00449 +MOVJ EC00449
SMOVL C00450 +MOVJ EC00450
SMOVL C00451 +MOVJ EC00451
SMOVL C00452 +MOVJ EC00452
SMOVL C00453 +MOVJ EC00453
SMOVL C00454 +MOVJ EC00454
SMOVL C00455 +MOVJ EC00455
SMOVL C00456 +MOVJ EC00456
SMOVL C00457 +MOVJ EC00457
SMOVL C00458 +MOVJ EC00458
SMOVL C00459 +MOVJ EC00459
SMOVL C00460 +MOVJ EC00460
SMOVL C00461 +MOVJ EC00461
SMOVL C00462 +MOVJ EC00462
SMOVL C00463 +MOVJ EC00463
SMOVL C00464 +MOVJ EC00464
SMOVL C00465 +MOVJ EC00465
SMOVL C00466 +MOVJ EC00466
SMOVL C00467 +MOVJ EC00467
SMOVL C00468 +MOVJ EC00468
SMOVL C00469 +MOVJ EC00469
SMOVL C00470 +MOVJ EC00470
SMOVL C00471 +MOVJ EC00471
SMOVL C00472 +MOVJ EC00472
SMOVL C00473 +MOVJ EC00473
SMOVL C00474 +MOVJ EC00474
SMOVL C00475 +MOVJ EC00475
SMOVL C00476 +MOVJ EC00476
SMOVL C00477 +MOVJ EC00477
SMOVL C00478 +MOVJ EC00478
SMOVL C00479 +MOVJ EC00479
SMOVL C00480 +MOVJ EC00480
SMOVL C00481 +MOVJ EC00481
SMOVL C00482 +MOVJ EC00482
SMOVL C00483 +MOVJ EC00483
SMOVL C00484 +MOVJ EC00484
SMOVL C00485 +MOVJ EC00485
SMOVL C00486 +MOVJ EC00486
SMOVL C00487 +MOVJ EC00487
SMOVL C00488 +MOVJ EC00488
SMOVL C00489 +MOVJ EC00489
SMOVL C00490 +MOVJ EC00490
SMOVL C00491 +MOVJ EC00491
SMOVL C00492 +MOVJ EC00492
SMOVL C00493 +MOVJ EC00493
SMOVL C00494 +MOVJ EC00494
SMOVL C00495 +MOVJ EC00495
SMOVL C00496 +MOVJ EC00496
SMOVL C00497 +MOVJ EC00497
SMOVL C00498 +MOVJ EC00498
SMOVL C00499 +MOVJ EC00499
SMOVL C00500 +MOVJ EC00500
SMOVL C00501 +MOVJ EC00501
SMOVL C00502 +MOVJ EC00502
SMOVL C00503 +MOVJ EC00503
SMOVL C00504 +MOVJ EC00504
SMOVL C00505 +MOVJ EC00505
SMOVL C00506 +MOVJ EC00506
SMOVL C00507 +MOVJ EC00507
SMOVL C00508 +MOVJ EC00508
SMOVL C00509 +MOVJ EC00509
SMOVL C00510 +MOVJ EC00510
SMOVL C00511 +MOVJ EC00511
SMOVL C00512 +MOVJ EC00512
SMOVL C00513 +MOVJ EC00513
SMOVL C00514 +MOVJ EC00514
SMOVL C00515 +MOVJ EC00515
SMOVL C00516 +MOVJ EC00516
SMOVL C00517 +MOVJ EC00517
SMOVL C00518 +MOVJ EC00518
SMOVL C00519 +MOVJ EC00519
SMOVL C00520 +MOVJ EC00520
SMOVL C00521 +MOVJ EC00521
SMOVL C00522 +MOVJ EC00522
SMOVL C00523 +MOVJ EC00523
SMOVL C00524 +MOVJ EC00524
SMOVL C00525 +MOVJ EC00525
SMOVL C00526 +MOVJ EC00526
SMOVL C00527 +MOVJ EC00527
SMOVL C00528 +MOVJ EC00528
SMOVL C00529 +MOVJ EC00529
SMOVL C00530 +MOVJ EC00530
SMOVL C00531 +MOVJ EC00531
SMOVL C00532 +MOVJ EC00532
SMOVL C00533 +MOVJ EC00533
SMOVL C00534 +MOVJ EC00534
SMOVL C00535 +MOVJ EC00535
SMOVL C00536 +MOVJ EC00536
SMOVL C00537 +MOVJ EC00537
SMOVL C00538 +MOVJ EC00538
SMOVL C00539 +MOVJ EC00539
SMOVL C00540 +MOVJ EC00540
SMOVL C00541 +MOVJ EC00541
SMOVL C00542 +MOVJ EC00542
SMOVL C00543 +MOVJ EC00543
SMOVL C00544 +MOVJ EC00544
SMOVL C00545 +MOVJ EC00545
SMOVL C00546 +MOVJ EC00546
SMOVL C00547 +MOVJ EC00547
SMOVL C00548 +MOVJ EC00548
SMOVL C00549 +MOVJ EC00549
SMOVL C00550 +MOVJ EC00550
SMOVL C00551 +MOVJ EC00551
SMOVL C00552 +MOVJ EC00552
SMOVL C00553 +MOVJ EC00553
SMOVL C00554 +MOVJ EC00554
SMOVL C00555 +MOVJ EC00555
SMOVL C00556 +MOVJ EC00556
SMOVL C00557 +MOVJ EC00557
SMOVL C00558 +MOVJ EC00558
SMOVL C00559 +MOVJ EC00559
SMOVL C00560 +MOVJ EC00560
SMOVL C00561 +MOVJ EC00561
SMOVL C00562 +MOVJ EC00562
SMOVL C00563 +MOVJ EC00563
SMOVL C00564 +MOVJ EC00564
SMOVL C00565 +MOVJ EC00565
SMOVL C00566 +MOVJ EC00566
SMOVL C00567 +MOVJ EC00567
SMOVL C00568 +MOVJ EC00568
SMOVL C00569 +MOVJ EC00569
SMOVL C00570 +MOVJ EC00570
SMOVL C00571 +MOVJ EC00571
SMOVL C00572 +MOVJ EC00572
SMOVL C00573 +MOVJ EC00573
SMOVL C00574 +MOVJ EC00574
SMOVL C00575 +MOVJ EC00575
SMOVL C00576 +MOVJ EC00576
SMOVL C00577 +MOVJ EC00577
SMOVL C00578 +MOVJ EC00578
SMOVL C00579 +MOVJ EC00579
SMOVL C00580 +MOVJ EC00580
SMOVL C00581 +MOVJ EC00581
SMOVL C00582 +MOVJ EC00582
SMOVL C00583 +MOVJ EC00583
SMOVL C00584 +MOVJ EC00584
SMOVL C00585 +MOVJ EC00585
SMOVL C00586 +MOVJ EC00586
SMOVL C00587 +MOVJ EC00587
SMOVL C00588 +MOVJ EC00588
SMOVL C00589 +MOVJ EC00589
SMOVL C00590 +MOVJ EC00590
SMOVL C00591 +MOVJ EC00591
SMOVL C00592 +MOVJ EC00592
SMOVL C00593 +MOVJ EC00593
SMOVL C00594 +MOVJ EC00594
SMOVL C00595 +MOVJ EC00595
SMOVL C00596 +MOVJ EC00596
SMOVL C00597 +MOVJ EC00597
SMOVL C00598 +MOVJ EC00598
SMOVL C00599 +MOVJ EC00599
SMOVL C00600 +MOVJ EC00600
SMOVL C00601 +MOVJ EC00601
SMOVL C00602 +MOVJ EC00602
SMOVL C00603 +MOVJ EC00603
SMOVL C00604 +MOVJ EC00604
SMOVL C00605 +MOVJ EC00605
SMOVL C00606 +MOVJ EC00606
SMOVL C00607 +MOVJ EC00607
SMOVL C00608 +MOVJ EC00608
SMOVL C00609 +MOVJ EC00609
SMOVL C00610 +MOVJ EC00610
SMOVL C00611 +MOVJ EC00611
SMOVL C00612 +MOVJ EC00612
SMOVL C00613 +MOVJ EC00613
SMOVL C00614 +MOVJ EC00614
SMOVL C00615 +MOVJ EC00615
SMOVL C00616 +MOVJ EC00616
SMOVL C00617 +MOVJ EC00617
SMOVL C00618 +MOVJ EC00618
SMOVL C00619 +MOVJ EC00619
SMOVL C00620 +MOVJ EC00620
SMOVL C00621 +MOVJ EC00621
SMOVL C00622 +MOVJ EC00622
SMOVL C00623 +MOVJ EC00623
SMOVL C00624 +MOVJ EC00624
SMOVL C00625 +MOVJ EC00625
SMOVL C00626 +MOVJ EC00626
SMOVL C00627 +MOVJ EC00627
SMOVL C00628 +MOVJ EC00628
SMOVL C00629 +MOVJ EC00629
SMOVL C00630 +MOVJ EC00630
SMOVL C00631 +MOVJ EC00631
SMOVL C00632 +MOVJ EC00632
SMOVL C00633 +MOVJ EC00633
SMOVL C00634 +MOVJ EC00634
SMOVL C00635 +MOVJ EC00635
SMOVL C00636 +MOVJ EC00636
SMOVL C00637 +MOVJ EC00637
SMOVL C00638 +MOVJ EC00638
SMOVL C00639 +MOVJ EC00639
SMOVL C00640 +MOVJ EC00640
SMOVL C00641 +MOVJ EC00641
SMOVL C00642 +MOVJ EC00642
SMOVL C00643 +MOVJ EC00643
SMOVL C00644 +MOVJ EC00644
SMOVL C00645 +MOVJ EC00645
SMOVL C00646 +MOVJ EC00646
SMOVL C00647 +MOVJ EC00647
SMOVL C00648 +MOVJ EC00648
SMOVL C00649 +MOVJ EC00649
SMOVL C00650 +MOVJ EC00650
SMOVL C00651 +MOVJ EC00651
SMOVL C00652 +MOVJ EC00652
SMOVL C00653 +MOVJ EC00653
SMOVL C00654 +MOVJ EC00654
SMOVL C00655 +MOVJ EC00655
SMOVL C00656 +MOVJ EC00656
SMOVL C00657 +MOVJ EC00657
SMOVL C00658 +MOVJ EC00658
SMOVL C00659 +MOVJ EC00659
SMOVL C00660 +MOVJ EC00660
SMOVL C00661 +MOVJ EC00661
SMOVL C00662 +MOVJ EC00662
SMOVL C00663 +MOVJ EC00663
SMOVL C00664 +MOVJ EC00664
SMOVL C00665 +MOVJ EC00665
SMOVL C00666 +MOVJ EC00666
SMOVL C00667 +MOVJ EC00667
SMOVL C00668 +MOVJ EC00668
SMOVL C00669 +MOVJ EC00669
SMOVL C00670 +MOVJ EC00670
SMOVL C00671 +MOVJ EC00671
SMOVL C00672 +MOVJ EC00672
SMOVL C00673 +MOVJ EC00673
SMOVL C00674 +MOVJ EC00674
SMOVL C00675 +MOVJ EC00675
SMOVL C00676 +MOVJ EC00676
SMOVL C00677 +MOVJ EC00677
SMOVL C00678 +MOVJ EC00678
SMOVL C00679 +MOVJ EC00679
SMOVL C00680 +MOVJ EC00680
SMOVL C00681 +MOVJ EC00681
SMOVL C00682 +MOVJ EC00682
SMOVL C00683 +MOVJ EC00683
SMOVL C00684 +MOVJ EC00684
SMOVL C00685 +MOVJ EC00685
SMOVL C00686 +MOVJ EC00686
SMOVL C00687 +MOVJ EC00687
SMOVL C00688 +MOVJ EC00688
SMOVL C00689 +MOVJ EC00689
SMOVL C00690 +MOVJ EC00690
SMOVL C00691 +MOVJ EC00691
SMOVL C00692 +MOVJ EC00692
SMOVL C00693 +MOVJ EC00693
SMOVL C00694 +MOVJ EC00694
SMOVL C00695 +MOVJ EC00695
SMOVL C00696 +MOVJ EC00696
SMOVL C00697 +MOVJ EC00697
SMOVL C00698 +MOVJ EC00698
SMOVL C00699 +MOVJ EC00699
SMOVL C00700 +MOVJ EC00700
SMOVL C00701 +MOVJ EC00701
SMOVL C00702 +MOVJ EC00702
SMOVL C00703 +MOVJ EC00703
SMOVL C00704 +MOVJ EC00704
SMOVL C00705 +MOVJ EC00705
SMOVL C00706 +MOVJ EC00706
SMOVL C00707 +MOVJ EC00707
SMOVL C00708 +MOVJ EC00708
SMOVL C00709 +MOVJ EC00709
SMOVL C00710 +MOVJ EC00710
SMOVL C00711 +MOVJ EC00711
SMOVL C00712 +MOVJ EC00712
SMOVL C00713 +MOVJ EC00713
SMOVL C00714 +MOVJ EC00714
SMOVL C00715 +MOVJ EC00715
SMOVL C00716 +MOVJ EC00716
SMOVL C00717 +MOVJ EC00717
SMOVL C00718 +MOVJ EC00718
SMOVL C00719 +MOVJ EC00719
SMOVL C00720 +MOVJ EC00720
SMOVL C00721 +MOVJ EC00721
SMOVL C00722 +MOVJ EC00722
SMOVL C00723 +MOVJ EC00723
SMOVL C00724 +MOVJ EC00724
SMOVL C00725 +MOVJ EC00725
SMOVL C00726 +MOVJ EC00726
SMOVL C00727 +MOVJ EC00727
SMOVL C00728 +MOVJ EC00728
SMOVL C00729 +MOVJ EC00729
SMOVL C00730 +MOVJ EC00730
SMOVL C00731 +MOVJ EC00731
SMOVL C00732 +MOVJ EC00732
SMOVL C00733 +MOVJ EC00733
SMOVL C00734 +MOVJ EC00734
SMOVL C00735 +MOVJ EC00735
SMOVL C00736 +MOVJ EC00736
SMOVL C00737 +MOVJ EC00737
SMOVL C00738 +MOVJ EC00738
SMOVL C00739 +MOVJ EC00739
SMOVL C00740 +MOVJ EC00740
SMOVL C00741 +MOVJ EC00741
SMOVL C00742 +MOVJ EC00742
SMOVL C00743 +MOVJ EC00743
SMOVL C00744 +MOVJ EC00744
SMOVL C00745 +MOVJ EC00745
SMOVL C00746 +MOVJ EC00746
SMOVL C00747 +MOVJ EC00747
SMOVL C00748 +MOVJ EC00748
SMOVL C00749 +MOVJ EC00749
SMOVL C00750 +MOVJ EC00750
SMOVL C00751 +MOVJ EC00751
SMOVL C00752 +MOVJ EC00752
SMOVL C00753 +MOVJ EC00753
SMOVL C00754 +MOVJ EC00754
SMOVL C00755 +MOVJ EC00755
SMOVL C00756 +MOVJ EC00756
SMOVL C00757 +MOVJ EC00757
SMOVL C00758 +MOVJ EC00758
SMOVL C00759 +MOVJ EC00759
SMOVL C00760 +MOVJ EC00760
SMOVL C00761 +MOVJ EC00761
SMOVL C00762 +MOVJ EC00762
SMOVL C00763 +MOVJ EC00763
SMOVL C00764 +MOVJ EC00764
SMOVL C00765 +MOVJ EC00765
SMOVL C00766 +MOVJ EC00766
SMOVL C00767 +MOVJ EC00767
SMOVL C00768 +MOVJ EC00768
SMOVL C00769 +MOVJ EC00769
SMOVL C00770 +MOVJ EC00770
SMOVL C00771 +MOVJ EC00771
SMOVL C00772 +MOVJ EC00772
SMOVL C00773 +MOVJ EC00773
SMOVL C00774 +MOVJ EC00774
SMOVL C00775 +MOVJ EC00775
SMOVL C00776 +MOVJ EC00776
SMOVL C00777 +MOVJ EC00777
SMOVL C00778 +MOVJ EC00778
SMOVL C00779 +MOVJ EC00779
SMOVL C00780 +MOVJ EC00780
SMOVL C00781 +MOVJ EC00781
SMOVL C00782 +MOVJ EC00782
SMOVL C00783 +MOVJ EC00783
SMOVL C00784 +MOVJ EC00784
SMOVL C00785 +MOVJ EC00785
SMOVL C00786 +MOVJ EC00786
SMOVL C00787 +MOVJ EC00787
SMOVL C00788 +MOVJ EC00788
SMOVL C00789 +MOVJ EC00789
SMOVL C00790 +MOVJ EC00790
SMOVL C00791 +MOVJ EC00791
SMOVL C00792 +MOVJ EC00792
SMOVL C00793 +MOVJ EC00793
SMOVL C00794 +MOVJ EC00794
SMOVL C00795 +MOVJ EC00795
SMOVL C00796 +MOVJ EC00796
SMOVL C00797 +MOVJ EC00797
SMOVL C00798 +MOVJ EC00798
SMOVL C00799 +MOVJ EC00799
SMOVL C00800 +MOVJ EC00800
SMOVL C00801 +MOVJ EC00801
SMOVL C00802 +MOVJ EC00802
SMOVL C00803 +MOVJ EC00803
SMOVL C00804 +MOVJ EC00804
SMOVL C00805 +MOVJ EC00805
SMOVL C00806 +MOVJ EC00806
SMOVL C00807 +MOVJ EC00807
SMOVL C00808 +MOVJ EC00808
SMOVL C00809 +MOVJ EC00809
SMOVL C00810 +MOVJ EC00810
SMOVL C00811 +MOVJ EC00811
SMOVL C00812 +MOVJ EC00812
SMOVL C00813 +MOVJ EC00813
SMOVL C00814 +MOVJ EC00814
SMOVL C00815 +MOVJ EC00815
SMOVL C00816 +MOVJ EC00816
SMOVL C00817 +MOVJ EC00817
SMOVL C00818 +MOVJ EC00818
SMOVL C00819 +MOVJ EC00819
SMOVL C00820 +MOVJ EC00820
SMOVL C00821 +MOVJ EC00821
SMOVL C00822 +MOVJ EC00822
SMOVL C00823 +MOVJ EC00823
SMOVL C00824 +MOVJ EC00824
SMOVL C00825 +MOVJ EC00825
SMOVL C00826 +MOVJ EC00826
SMOVL C00827 +MOVJ EC00827
SMOVL C00828 +MOVJ EC00828
SMOVL C00829 +MOVJ EC00829
SMOVL C00830 +MOVJ EC00830
SMOVL C00831 +MOVJ EC00831
SMOVL C00832 +MOVJ EC00832
SMOVL C00833 +MOVJ EC00833
SMOVL C00834 +MOVJ EC00834
SMOVL C00835 +MOVJ EC00835
SMOVL C00836 +MOVJ EC00836
SMOVL C00837 +MOVJ EC00837
SMOVL C00838 +MOVJ EC00838
SMOVL C00839 +MOVJ EC00839
SMOVL C00840 +MOVJ EC00840
SMOVL C00841 +MOVJ EC00841
SMOVL C00842 +MOVJ EC00842
SMOVL C00843 +MOVJ EC00843
SMOVL C00844 +MOVJ EC00844
SMOVL C00845 +MOVJ EC00845
SMOVL C00846 +MOVJ EC00846
SMOVL C00847 +MOVJ EC00847
SMOVL C00848 +MOVJ EC00848
SMOVL C00849 +MOVJ EC00849
SMOVL C00850 +MOVJ EC00850
SMOVL C00851 +MOVJ EC00851
SMOVL C00852 +MOVJ EC00852
SMOVL C00853 +MOVJ EC00853
SMOVL C00854 +MOVJ EC00854
SMOVL C00855 +MOVJ EC00855
SMOVL C00856 +MOVJ EC00856
SMOVL C00857 +MOVJ EC00857
SMOVL C00858 +MOVJ EC00858
SMOVL C00859 +MOVJ EC00859
SMOVL C00860 +MOVJ EC00860
SMOVL C00861 +MOVJ EC00861
SMOVL C00862 +MOVJ EC00862
SMOVL C00863 +MOVJ EC00863
SMOVL C00864 +MOVJ EC00864
SMOVL C00865 +MOVJ EC00865
SMOVL C00866 +MOVJ EC00866
SMOVL C00867 +MOVJ EC00867
SMOVL C00868 +MOVJ EC00868
SMOVL C00869 +MOVJ EC00869
SMOVL C00870 +MOVJ EC00870
SMOVL C00871 +MOVJ EC00871
SMOVL C00872 +MOVJ EC00872
SMOVL C00873 +MOVJ EC00873
SMOVL C00874 +MOVJ EC00874
SMOVL C00875 +MOVJ EC00875
SMOVL C00876 +MOVJ EC00876
SMOVL C00877 +MOVJ EC00877
SMOVL C00878 +MOVJ EC00878
SMOVL C00879 +MOVJ EC00879
SMOVL C00880 +MOVJ EC00880
SMOVL C00881 +MOVJ EC00881
SMOVL C00882 +MOVJ EC00882
SMOVL C00883 +MOVJ EC00883
SMOVL C00884 +MOVJ EC00884
SMOVL C00885 +MOVJ EC00885
SMOVL C00886 +MOVJ EC00886
SMOVL C00887 +MOVJ EC00887
SMOVL C00888 +MOVJ EC00888
SMOVL C00889 +MOVJ EC00889
SMOVL C00890 +MOVJ EC00890
SMOVL C00891 +MOVJ EC00891
SMOVL C00892 +MOVJ EC00892
SMOVL C00893 +MOVJ EC00893
SMOVL C00894 +MOVJ EC00894
SMOVL C00895 +MOVJ EC00895
SMOVL C00896 +MOVJ EC00896
SMOVL C00897 +MOVJ EC00897
SMOVL C00898 +MOVJ EC00898
ARCOF
SMOVL C00899 +MOVJ EC00899
ARCON
SMOVL C00900 +MOVJ EC00900
SMOVL C00901 +MOVJ EC00901
SMOVL C00902 +MOVJ EC00902
SMOVL C00903 +MOVJ EC00903
SMOVL C00904 +MOVJ EC00904
SMOVL C00905 +MOVJ EC00905
SMOVL C00906 +MOVJ EC00906
SMOVL C00907 +MOVJ EC00907
SMOVL C00908 +MOVJ EC00908
SMOVL C00909 +MOVJ EC00909
SMOVL C00910 +MOVJ EC00910
SMOVL C00911 +MOVJ EC00911
SMOVL C00912 +MOVJ EC00912
SMOVL C00913 +MOVJ EC00913
SMOVL C00914 +MOVJ EC00914
SMOVL C00915 +MOVJ EC00915
SMOVL C00916 +MOVJ EC00916
SMOVL C00917 +MOVJ EC00917
ARCOF
SMOVL C00918 +MOVJ EC00918
ARCON
SMOVL C00919 +MOVJ EC00919
SMOVL C00920 +MOVJ EC00920
SMOVL C00921 +MOVJ EC00921
SMOVL C00922 +MOVJ EC00922
SMOVL C00923 +MOVJ EC00923
SMOVL C00924 +MOVJ EC00924
SMOVL C00925 +MOVJ EC00925
SMOVL C00926 +MOVJ EC00926
SMOVL C00927 +MOVJ EC00927
SMOVL C00928 +MOVJ EC00928
SMOVL C00929 +MOVJ EC00929
SMOVL C00930 +MOVJ EC00930
SMOVL C00931 +MOVJ EC00931
SMOVL C00932 +MOVJ EC00932
SMOVL C00933 +MOVJ EC00933
SMOVL C00934 +MOVJ EC00934
SMOVL C00935 +MOVJ EC00935
SMOVL C00936 +MOVJ EC00936
ARCOF
SMOVL C00937 +MOVJ EC00937
ARCON
SMOVL C00938 +MOVJ EC00938
SMOVL C00939 +MOVJ EC00939
SMOVL C00940 +MOVJ EC00940
SMOVL C00941 +MOVJ EC00941
SMOVL C00942 +MOVJ EC00942
SMOVL C00943 +MOVJ EC00943
SMOVL C00944 +MOVJ EC00944
SMOVL C00945 +MOVJ EC00945
SMOVL C00946 +MOVJ EC00946
SMOVL C00947 +MOVJ EC00947
SMOVL C00948 +MOVJ EC00948
SMOVL C00949 +MOVJ EC00949
SMOVL C00950 +MOVJ EC00950
SMOVL C00951 +MOVJ EC00951
SMOVL C00952 +MOVJ EC00952
SMOVL C00953 +MOVJ EC00953
SMOVL C00954 +MOVJ EC00954
SMOVL C00955 +MOVJ EC00955
ARCOF
SMOVL C00956 +MOVJ EC00956
ARCON
SMOVL C00957 +MOVJ EC00957
SMOVL C00958 +MOVJ EC00958
SMOVL C00959 +MOVJ EC00959
SMOVL C00960 +MOVJ EC00960
SMOVL C00961 +MOVJ EC00961
SMOVL C00962 +MOVJ EC00962
SMOVL C00963 +MOVJ EC00963
SMOVL C00964 +MOVJ EC00964
SMOVL C00965 +MOVJ EC00965
SMOVL C00966 +MOVJ EC00966
SMOVL C00967 +MOVJ EC00967
SMOVL C00968 +MOVJ EC00968
SMOVL C00969 +MOVJ EC00969
SMOVL C00970 +MOVJ EC00970
SMOVL C00971 +MOVJ EC00971
SMOVL C00972 +MOVJ EC00972
SMOVL C00973 +MOVJ EC00973
SMOVL C00974 +MOVJ EC00974
SMOVL C00975 +MOVJ EC00975
ARCOF
SMOVL C00976 +MOVJ EC00976
ARCON
SMOVL C00977 +MOVJ EC00977
SMOVL C00978 +MOVJ EC00978
SMOVL C00979 +MOVJ EC00979
SMOVL C00980 +MOVJ EC00980
SMOVL C00981 +MOVJ EC00981
SMOVL C00982 +MOVJ EC00982
SMOVL C00983 +MOVJ EC00983
SMOVL C00984 +MOVJ EC00984
SMOVL C00985 +MOVJ EC00985
SMOVL C00986 +MOVJ EC00986
SMOVL C00987 +MOVJ EC00987
SMOVL C00988 +MOVJ EC00988
SMOVL C00989 +MOVJ EC00989
SMOVL C00990 +MOVJ EC00990
SMOVL C00991 +MOVJ EC00991
SMOVL C00992 +MOVJ EC00992
SMOVL C00993 +MOVJ EC00993
SMOVL C00994 +MOVJ EC00994
ARCOF
SMOVL C00995 +MOVJ EC00995
ARCON
SMOVL C00996 +MOVJ EC00996
SMOVL C00997 +MOVJ EC00997
SMOVL C00998 +MOVJ EC00998
SMOVL C00999 +MOVJ EC00999
SMOVL C01000 +MOVJ EC01000
SMOVL C01001 +MOVJ EC01001
SMOVL C01002 +MOVJ EC01002
SMOVL C01003 +MOVJ EC01003
SMOVL C01004 +MOVJ EC01004
SMOVL C01005 +MOVJ EC01005
SMOVL C01006 +MOVJ EC01006
SMOVL C01007 +MOVJ EC01007
SMOVL C01008 +MOVJ EC01008
SMOVL C01009 +MOVJ EC01009
SMOVL C01010 +MOVJ EC01010
SMOVL C01011 +MOVJ EC01011
SMOVL C01012 +MOVJ EC01012
SMOVL C01013 +MOVJ EC01013
ARCOF
SMOVL C01014 +MOVJ EC01014
ARCON
SMOVL C01015 +MOVJ EC01015
SMOVL C01016 +MOVJ EC01016
SMOVL C01017 +MOVJ EC01017
SMOVL C01018 +MOVJ EC01018
SMOVL C01019 +MOVJ EC01019
SMOVL C01020 +MOVJ EC01020
SMOVL C01021 +MOVJ EC01021
SMOVL C01022 +MOVJ EC01022
SMOVL C01023 +MOVJ EC01023
SMOVL C01024 +MOVJ EC01024
SMOVL C01025 +MOVJ EC01025
SMOVL C01026 +MOVJ EC01026
SMOVL C01027 +MOVJ EC01027
SMOVL C01028 +MOVJ EC01028
SMOVL C01029 +MOVJ EC01029
SMOVL C01030 +MOVJ EC01030
SMOVL C01031 +MOVJ EC01031
SMOVL C01032 +MOVJ EC01032
ARCOF
SMOVL C01033 +MOVJ EC01033
ARCON
SMOVL C01034 +MOVJ EC01034
SMOVL C01035 +MOVJ EC01035
SMOVL C01036 +MOVJ EC01036
SMOVL C01037 +MOVJ EC01037
SMOVL C01038 +MOVJ EC01038
SMOVL C01039 +MOVJ EC01039
SMOVL C01040 +MOVJ EC01040
SMOVL C01041 +MOVJ EC01041
SMOVL C01042 +MOVJ EC01042
SMOVL C01043 +MOVJ EC01043
SMOVL C01044 +MOVJ EC01044
SMOVL C01045 +MOVJ EC01045
SMOVL C01046 +MOVJ EC01046
SMOVL C01047 +MOVJ EC01047
SMOVL C01048 +MOVJ EC01048
SMOVL C01049 +MOVJ EC01049
ARCOF
SMOVL C01050 +MOVJ EC01050
ARCON
SMOVL C01051 +MOVJ EC01051
SMOVL C01052 +MOVJ EC01052
SMOVL C01053 +MOVJ EC01053
SMOVL C01054 +MOVJ EC01054
SMOVL C01055 +MOVJ EC01055
SMOVL C01056 +MOVJ EC01056
SMOVL C01057 +MOVJ EC01057
SMOVL C01058 +MOVJ EC01058
SMOVL C01059 +MOVJ EC01059
SMOVL C01060 +MOVJ EC01060
SMOVL C01061 +MOVJ EC01061
SMOVL C01062 +MOVJ EC01062
ARCOF
SMOVL C01063 +MOVJ EC01063
ARCON
SMOVL C01064 +MOVJ EC01064
SMOVL C01065 +MOVJ EC01065
SMOVL C01066 +MOVJ EC01066
SMOVL C01067 +MOVJ EC01067
SMOVL C01068 +MOVJ EC01068
SMOVL C01069 +MOVJ EC01069
SMOVL C01070 +MOVJ EC01070
SMOVL C01071 +MOVJ EC01071
SMOVL C01072 +MOVJ EC01072
SMOVL C01073 +MOVJ EC01073
SMOVL C01074 +MOVJ EC01074
SMOVL C01075 +MOVJ EC01075
ARCOF
SMOVL C01076 +MOVJ EC01076
ARCON
SMOVL C01077 +MOVJ EC01077
SMOVL C01078 +MOVJ EC01078
SMOVL C01079 +MOVJ EC01079
SMOVL C01080 +MOVJ EC01080
SMOVL C01081 +MOVJ EC01081
SMOVL C01082 +MOVJ EC01082
SMOVL C01083 +MOVJ EC01083
SMOVL C01084 +MOVJ EC01084
SMOVL C01085 +MOVJ EC01085
SMOVL C01086 +MOVJ EC01086
SMOVL C01087 +MOVJ EC01087
SMOVL C01088 +MOVJ EC01088
ARCOF
SMOVL C01089 +MOVJ EC01089
ARCON
SMOVL C01090 +MOVJ EC01090
SMOVL C01091 +MOVJ EC01091
SMOVL C01092 +MOVJ EC01092
SMOVL C01093 +MOVJ EC01093
SMOVL C01094 +MOVJ EC01094
SMOVL C01095 +MOVJ EC01095
SMOVL C01096 +MOVJ EC01096
SMOVL C01097 +MOVJ EC01097
SMOVL C01098 +MOVJ EC01098
SMOVL C01099 +MOVJ EC01099
SMOVL C01100 +MOVJ EC01100
SMOVL C01101 +MOVJ EC01101
SMOVL C01102 +MOVJ EC01102
ARCOF
SMOVL C01103 +MOVJ EC01103
ARCON
SMOVL C01104 +MOVJ EC01104
SMOVL C01105 +MOVJ EC01105
SMOVL C01106 +MOVJ EC01106
SMOVL C01107 +MOVJ EC01107
SMOVL C01108 +MOVJ EC01108
SMOVL C01109 +MOVJ EC01109
SMOVL C01110 +MOVJ EC01110
SMOVL C01111 +MOVJ EC01111
SMOVL C01112 +MOVJ EC01112
SMOVL C01113 +MOVJ EC01113
SMOVL C01114 +MOVJ EC01114
SMOVL C01115 +MOVJ EC01115
ARCOF
SMOVL C01116 +MOVJ EC01116
ARCON
SMOVL C01117 +MOVJ EC01117
SMOVL C01118 +MOVJ EC01118
SMOVL C01119 +MOVJ EC01119
SMOVL C01120 +MOVJ EC01120
SMOVL C01121 +MOVJ EC01121
SMOVL C01122 +MOVJ EC01122
SMOVL C01123 +MOVJ EC01123
SMOVL C01124 +MOVJ EC01124
SMOVL C01125 +MOVJ EC01125
SMOVL C01126 +MOVJ EC01126
SMOVL C01127 +MOVJ EC01127
SMOVL C01128 +MOVJ EC01128
ARCOF
SMOVL C01129 +MOVJ EC01129
ARCON
SMOVL C01130 +MOVJ EC01130
SMOVL C01131 +MOVJ EC01131
SMOVL C01132 +MOVJ EC01132
SMOVL C01133 +MOVJ EC01133
SMOVL C01134 +MOVJ EC01134
SMOVL C01135 +MOVJ EC01135
SMOVL C01136 +MOVJ EC01136
SMOVL C01137 +MOVJ EC01137
SMOVL C01138 +MOVJ EC01138
SMOVL C01139 +MOVJ EC01139
SMOVL C01140 +MOVJ EC01140
SMOVL C01141 +MOVJ EC01141
ARCOF
SMOVL C01142 +MOVJ EC01142
ARCON
SMOVL C01143 +MOVJ EC01143
SMOVL C01144 +MOVJ EC01144
SMOVL C01145 +MOVJ EC01145
SMOVL C01146 +MOVJ EC01146
SMOVL C01147 +MOVJ EC01147
SMOVL C01148 +MOVJ EC01148
SMOVL C01149 +MOVJ EC01149
SMOVL C01150 +MOVJ EC01150
SMOVL C01151 +MOVJ EC01151
SMOVL C01152 +MOVJ EC01152
SMOVL C01153 +MOVJ EC01153
SMOVL C01154 +MOVJ EC01154
ARCOF
SMOVL C01155 +MOVJ EC01155
ARCON
SMOVL C01156 +MOVJ EC01156
SMOVL C01157 +MOVJ EC01157
SMOVL C01158 +MOVJ EC01158
SMOVL C01159 +MOVJ EC01159
SMOVL C01160 +MOVJ EC01160
SMOVL C01161 +MOVJ EC01161
SMOVL C01162 +MOVJ EC01162
SMOVL C01163 +MOVJ EC01163
SMOVL C01164 +MOVJ EC01164
SMOVL C01165 +MOVJ EC01165
ARCOF
SMOVL C01166 +MOVJ EC01166
ARCON
SMOVL C01167 +MOVJ EC01167
SMOVL C01168 +MOVJ EC01168
SMOVL C01169 +MOVJ EC01169
SMOVL C01170 +MOVJ EC01170
SMOVL C01171 +MOVJ EC01171
SMOVL C01172 +MOVJ EC01172
SMOVL C01173 +MOVJ EC01173
SMOVL C01174 +MOVJ EC01174
SMOVL C01175 +MOVJ EC01175
SMOVL C01176 +MOVJ EC01176
ARCOF
SMOVL C01177 +MOVJ EC01177
ARCON
SMOVL C01178 +MOVJ EC01178
SMOVL C01179 +MOVJ EC01179
SMOVL C01180 +MOVJ EC01180
SMOVL C01181 +MOVJ EC01181
SMOVL C01182 +MOVJ EC01182
SMOVL C01183 +MOVJ EC01183
SMOVL C01184 +MOVJ EC01184
SMOVL C01185 +MOVJ EC01185
SMOVL C01186 +MOVJ EC01186
SMOVL C01187 +MOVJ EC01187
ARCOF
SMOVL C01188 +MOVJ EC01188
ARCON
SMOVL C01189 +MOVJ EC01189
SMOVL C01190 +MOVJ EC01190
SMOVL C01191 +MOVJ EC01191
SMOVL C01192 +MOVJ EC01192
SMOVL C01193 +MOVJ EC01193
SMOVL C01194 +MOVJ EC01194
SMOVL C01195 +MOVJ EC01195
SMOVL C01196 +MOVJ EC01196
SMOVL C01197 +MOVJ EC01197
SMOVL C01198 +MOVJ EC01198
SMOVL C01199 +MOVJ EC01199
ARCOF
SMOVL C01200 +MOVJ EC01200
ARCON
SMOVL C01201 +MOVJ EC01201
SMOVL C01202 +MOVJ EC01202
SMOVL C01203 +MOVJ EC01203
SMOVL C01204 +MOVJ EC01204
SMOVL C01205 +MOVJ EC01205
SMOVL C01206 +MOVJ EC01206
SMOVL C01207 +MOVJ EC01207
SMOVL C01208 +MOVJ EC01208
SMOVL C01209 +MOVJ EC01209
SMOVL C01210 +MOVJ EC01210
ARCOF
SMOVL C01211 +MOVJ EC01211
ARCON
SMOVL C01212 +MOVJ EC01212
SMOVL C01213 +MOVJ EC01213
SMOVL C01214 +MOVJ EC01214
SMOVL C01215 +MOVJ EC01215
SMOVL C01216 +MOVJ EC01216
SMOVL C01217 +MOVJ EC01217
SMOVL C01218 +MOVJ EC01218
SMOVL C01219 +MOVJ EC01219
SMOVL C01220 +MOVJ EC01220
SMOVL C01221 +MOVJ EC01221
ARCOF
SMOVL C01222 +MOVJ EC01222
ARCON
SMOVL C01223 +MOVJ EC01223
SMOVL C01224 +MOVJ EC01224
SMOVL C01225 +MOVJ EC01225
SMOVL C01226 +MOVJ EC01226
SMOVL C01227 +MOVJ EC01227
SMOVL C01228 +MOVJ EC01228
SMOVL C01229 +MOVJ EC01229
SMOVL C01230 +MOVJ EC01230
SMOVL C01231 +MOVJ EC01231
SMOVL C01232 +MOVJ EC01232
ARCOF
SMOVL C01233 +MOVJ EC01233
ARCON
SMOVL C01234 +MOVJ EC01234
SMOVL C01235 +MOVJ EC01235
SMOVL C01236 +MOVJ EC01236
SMOVL C01237 +MOVJ EC01237
SMOVL C01238 +MOVJ EC01238
SMOVL C01239 +MOVJ EC01239
SMOVL C01240 +MOVJ EC01240
SMOVL C01241 +MOVJ EC01241
SMOVL C01242 +MOVJ EC01242
SMOVL C01243 +MOVJ EC01243
SMOVL C01244 +MOVJ EC01244
ARCOF
SMOVL C01245 +MOVJ EC01245
ARCON
SMOVL C01246 +MOVJ EC01246
SMOVL C01247 +MOVJ EC01247
SMOVL C01248 +MOVJ EC01248
SMOVL C01249 +MOVJ EC01249
SMOVL C01250 +MOVJ EC01250
SMOVL C01251 +MOVJ EC01251
SMOVL C01252 +MOVJ EC01252
SMOVL C01253 +MOVJ EC01253
SMOVL C01254 +MOVJ EC01254
SMOVL C01255 +MOVJ EC01255
ARCOF
SMOVL C01256 +MOVJ EC01256
ARCON
SMOVL C01257 +MOVJ EC01257
SMOVL C01258 +MOVJ EC01258
SMOVL C01259 +MOVJ EC01259
SMOVL C01260 +MOVJ EC01260
SMOVL C01261 +MOVJ EC01261
SMOVL C01262 +MOVJ EC01262
SMOVL C01263 +MOVJ EC01263
SMOVL C01264 +MOVJ EC01264
SMOVL C01265 +MOVJ EC01265
SMOVL C01266 +MOVJ EC01266
ARCOF
SMOVL C01267 +MOVJ EC01267
ARCON
SMOVL C01268 +MOVJ EC01268
SMOVL C01269 +MOVJ EC01269
SMOVL C01270 +MOVJ EC01270
SMOVL C01271 +MOVJ EC01271
SMOVL C01272 +MOVJ EC01272
SMOVL C01273 +MOVJ EC01273
SMOVL C01274 +MOVJ EC01274
SMOVL C01275 +MOVJ EC01275
SMOVL C01276 +MOVJ EC01276
SMOVL C01277 +MOVJ EC01277
ARCOF
SMOVL C01278 +MOVJ EC01278
ARCON
SMOVL C01279 +MOVJ EC01279
SMOVL C01280 +MOVJ EC01280
SMOVL C01281 +MOVJ EC01281
SMOVL C01282 +MOVJ EC01282
SMOVL C01283 +MOVJ EC01283
SMOVL C01284 +MOVJ EC01284
SMOVL C01285 +MOVJ EC01285
SMOVL C01286 +MOVJ EC01286
SMOVL C01287 +MOVJ EC01287
SMOVL C01288 +MOVJ EC01288
SMOVL C01289 +MOVJ EC01289
ARCOF
SMOVL C01290 +MOVJ EC01290
ARCON
SMOVL C01291 +MOVJ EC01291
SMOVL C01292 +MOVJ EC01292
SMOVL C01293 +MOVJ EC01293
SMOVL C01294 +MOVJ EC01294
SMOVL C01295 +MOVJ EC01295
SMOVL C01296 +MOVJ EC01296
SMOVL C01297 +MOVJ EC01297
SMOVL C01298 +MOVJ EC01298
SMOVL C01299 +MOVJ EC01299
SMOVL C01300 +MOVJ EC01300
ARCOF
SMOVL C01301 +MOVJ EC01301
ARCON
SMOVL C01302 +MOVJ EC01302
SMOVL C01303 +MOVJ EC01303
SMOVL C01304 +MOVJ EC01304
SMOVL C01305 +MOVJ EC01305
SMOVL C01306 +MOVJ EC01306
SMOVL C01307 +MOVJ EC01307
SMOVL C01308 +MOVJ EC01308
SMOVL C01309 +MOVJ EC01309
SMOVL C01310 +MOVJ EC01310
SMOVL C01311 +MOVJ EC01311
ARCOF
SMOVL C01312 +MOVJ EC01312
ARCON
SMOVL C01313 +MOVJ EC01313
SMOVL C01314 +MOVJ EC01314
SMOVL C01315 +MOVJ EC01315
SMOVL C01316 +MOVJ EC01316
SMOVL C01317 +MOVJ EC01317
SMOVL C01318 +MOVJ EC01318
SMOVL C01319 +MOVJ EC01319
SMOVL C01320 +MOVJ EC01320
SMOVL C01321 +MOVJ EC01321
SMOVL C01322 +MOVJ EC01322
ARCOF
SMOVL C01323 +MOVJ EC01323
ARCON
SMOVL C01324 +MOVJ EC01324
SMOVL C01325 +MOVJ EC01325
SMOVL C01326 +MOVJ EC01326
SMOVL C01327 +MOVJ EC01327
SMOVL C01328 +MOVJ EC01328
SMOVL C01329 +MOVJ EC01329
SMOVL C01330 +MOVJ EC01330
SMOVL C01331 +MOVJ EC01331
SMOVL C01332 +MOVJ EC01332
SMOVL C01333 +MOVJ EC01333
ARCOF
SMOVL C01334 +MOVJ EC01334
ARCON
SMOVL C01335 +MOVJ EC01335
SMOVL C01336 +MOVJ EC01336
SMOVL C01337 +MOVJ EC01337
SMOVL C01338 +MOVJ EC01338
SMOVL C01339 +MOVJ EC01339
SMOVL C01340 +MOVJ EC01340
SMOVL C01341 +MOVJ EC01341
SMOVL C01342 +MOVJ EC01342
ARCOF
SMOVL C01343 +MOVJ EC01343
ARCON
SMOVL C01344 +MOVJ EC01344
SMOVL C01345 +MOVJ EC01345
SMOVL C01346 +MOVJ EC01346
SMOVL C01347 +MOVJ EC01347
SMOVL C01348 +MOVJ EC01348
SMOVL C01349 +MOVJ EC01349
SMOVL C01350 +MOVJ EC01350
SMOVL C01351 +MOVJ EC01351
ARCOF
SMOVL C01352 +MOVJ EC01352
ARCON
SMOVL C01353 +MOVJ EC01353
SMOVL C01354 +MOVJ EC01354
SMOVL C01355 +MOVJ EC01355
SMOVL C01356 +MOVJ EC01356
SMOVL C01357 +MOVJ EC01357
SMOVL C01358 +MOVJ EC01358
SMOVL C01359 +MOVJ EC01359
SMOVL C01360 +MOVJ EC01360
ARCOF
SMOVL C01361 +MOVJ EC01361
ARCON
SMOVL C01362 +MOVJ EC01362
SMOVL C01363 +MOVJ EC01363
SMOVL C01364 +MOVJ EC01364
SMOVL C01365 +MOVJ EC01365
SMOVL C01366 +MOVJ EC01366
SMOVL C01367 +MOVJ EC01367
SMOVL C01368 +MOVJ EC01368
SMOVL C01369 +MOVJ EC01369
SMOVL C01370 +MOVJ EC01370
ARCOF
SMOVL C01371 +MOVJ EC01371
ARCON
SMOVL C01372 +MOVJ EC01372
SMOVL C01373 +MOVJ EC01373
SMOVL C01374 +MOVJ EC01374
SMOVL C01375 +MOVJ EC01375
SMOVL C01376 +MOVJ EC01376
SMOVL C01377 +MOVJ EC01377
SMOVL C01378 +MOVJ EC01378
SMOVL C01379 +MOVJ EC01379
ARCOF
SMOVL C01380 +MOVJ EC01380
ARCON
SMOVL C01381 +MOVJ EC01381
SMOVL C01382 +MOVJ EC01382
SMOVL C01383 +MOVJ EC01383
SMOVL C01384 +MOVJ EC01384
SMOVL C01385 +MOVJ EC01385
SMOVL C01386 +MOVJ EC01386
SMOVL C01387 +MOVJ EC01387
SMOVL C01388 +MOVJ EC01388
ARCOF
SMOVL C01389 +MOVJ EC01389
ARCON
SMOVL C01390 +MOVJ EC01390
SMOVL C01391 +MOVJ EC01391
SMOVL C01392 +MOVJ EC01392
SMOVL C01393 +MOVJ EC01393
SMOVL C01394 +MOVJ EC01394
SMOVL C01395 +MOVJ EC01395
SMOVL C01396 +MOVJ EC01396
SMOVL C01397 +MOVJ EC01397
ARCOF
SMOVL C01398 +MOVJ EC01398
ARCON
SMOVL C01399 +MOVJ EC01399
SMOVL C01400 +MOVJ EC01400
SMOVL C01401 +MOVJ EC01401
SMOVL C01402 +MOVJ EC01402
SMOVL C01403 +MOVJ EC01403
SMOVL C01404 +MOVJ EC01404
SMOVL C01405 +MOVJ EC01405
SMOVL C01406 +MOVJ EC01406
ARCOF
SMOVL C01407 +MOVJ EC01407
ARCON
SMOVL C01408 +MOVJ EC01408
SMOVL C01409 +MOVJ EC01409
SMOVL C01410 +MOVJ EC01410
SMOVL C01411 +MOVJ EC01411
SMOVL C01412 +MOVJ EC01412
SMOVL C01413 +MOVJ EC01413
ARCOF
SMOVL C01414 +MOVJ EC01414
ARCON
SMOVL C01415 +MOVJ EC01415
SMOVL C01416 +MOVJ EC01416
SMOVL C01417 +MOVJ EC01417
SMOVL C01418 +MOVJ EC01418
SMOVL C01419 +MOVJ EC01419
SMOVL C01420 +MOVJ EC01420
ARCOF
SMOVL C01421 +MOVJ EC01421
ARCON
SMOVL C01422 +MOVJ EC01422
SMOVL C01423 +MOVJ EC01423
SMOVL C01424 +MOVJ EC01424
SMOVL C01425 +MOVJ EC01425
SMOVL C01426 +MOVJ EC01426
SMOVL C01427 +MOVJ EC01427
ARCOF
SMOVL C01428 +MOVJ EC01428
ARCON
SMOVL C01429 +MOVJ EC01429
SMOVL C01430 +MOVJ EC01430
SMOVL C01431 +MOVJ EC01431
SMOVL C01432 +MOVJ EC01432
SMOVL C01433 +MOVJ EC01433
SMOVL C01434 +MOVJ EC01434
SMOVL C01435 +MOVJ EC01435
ARCOF
SMOVL C01436 +MOVJ EC01436
ARCON
SMOVL C01437 +MOVJ EC01437
SMOVL C01438 +MOVJ EC01438
SMOVL C01439 +MOVJ EC01439
SMOVL C01440 +MOVJ EC01440
SMOVL C01441 +MOVJ EC01441
SMOVL C01442 +MOVJ EC01442
ARCOF
SMOVL C01443 +MOVJ EC01443
ARCON
SMOVL C01444 +MOVJ EC01444
SMOVL C01445 +MOVJ EC01445
SMOVL C01446 +MOVJ EC01446
SMOVL C01447 +MOVJ EC01447
SMOVL C01448 +MOVJ EC01448
SMOVL C01449 +MOVJ EC01449
ARCOF
SMOVL C01450 +MOVJ EC01450
ARCON
SMOVL C01451 +MOVJ EC01451
SMOVL C01452 +MOVJ EC01452
SMOVL C01453 +MOVJ EC01453
SMOVL C01454 +MOVJ EC01454
SMOVL C01455 +MOVJ EC01455
SMOVL C01456 +MOVJ EC01456
ARCOF
SMOVL C01457 +MOVJ EC01457
ARCON
SMOVL C01458 +MOVJ EC01458
SMOVL C01459 +MOVJ EC01459
SMOVL C01460 +MOVJ EC01460
SMOVL C01461 +MOVJ EC01461
SMOVL C01462 +MOVJ EC01462
SMOVL C01463 +MOVJ EC01463
SMOVL C01464 +MOVJ EC01464
ARCOF
SMOVL C01465 +MOVJ EC01465
ARCON
SMOVL C01466 +MOVJ EC01466
SMOVL C01467 +MOVJ EC01467
SMOVL C01468 +MOVJ EC01468
SMOVL C01469 +MOVJ EC01469
SMOVL C01470 +MOVJ EC01470
SMOVL C01471 +MOVJ EC01471
ARCOF
SMOVL C01472 +MOVJ EC01472
ARCON
SMOVL C01473 +MOVJ EC01473
SMOVL C01474 +MOVJ EC01474
SMOVL C01475 +MOVJ EC01475
SMOVL C01476 +MOVJ EC01476
SMOVL C01477 +MOVJ EC01477
SMOVL C01478 +MOVJ EC01478
ARCOF
SMOVL C01479 +MOVJ EC01479
ARCON
SMOVL C01480 +MOVJ EC01480
SMOVL C01481 +MOVJ EC01481
SMOVL C01482 +MOVJ EC01482
SMOVL C01483 +MOVJ EC01483
SMOVL C01484 +MOVJ EC01484
SMOVL C01485 +MOVJ EC01485
ARCOF
SMOVL C01486 +MOVJ EC01486
ARCON
SMOVL C01487 +MOVJ EC01487
SMOVL C01488 +MOVJ EC01488
SMOVL C01489 +MOVJ EC01489
SMOVL C01490 +MOVJ EC01490
SMOVL C01491 +MOVJ EC01491
SMOVL C01492 +MOVJ EC01492
SMOVL C01493 +MOVJ EC01493
ARCOF
SMOVL C01494 +MOVJ EC01494
ARCON
SMOVL C01495 +MOVJ EC01495
SMOVL C01496 +MOVJ EC01496
SMOVL C01497 +MOVJ EC01497
SMOVL C01498 +MOVJ EC01498
SMOVL C01499 +MOVJ EC01499
SMOVL C01500 +MOVJ EC01500
ARCOF
SMOVL C01501 +MOVJ EC01501
ARCON
SMOVL C01502 +MOVJ EC01502
SMOVL C01503 +MOVJ EC01503
SMOVL C01504 +MOVJ EC01504
SMOVL C01505 +MOVJ EC01505
SMOVL C01506 +MOVJ EC01506
SMOVL C01507 +MOVJ EC01507
ARCOF
SMOVL C01508 +MOVJ EC01508
ARCON
SMOVL C01509 +MOVJ EC01509
SMOVL C01510 +MOVJ EC01510
SMOVL C01511 +MOVJ EC01511
SMOVL C01512 +MOVJ EC01512
SMOVL C01513 +MOVJ EC01513
SMOVL C01514 +MOVJ EC01514
ARCOF
SMOVL C01515 +MOVJ EC01515
ARCON
SMOVL C01516 +MOVJ EC01516
SMOVL C01517 +MOVJ EC01517
SMOVL C01518 +MOVJ EC01518
END
